(*
    Read and refresh axis parameters
*)
FUNCTION_BLOCK FB_ReadParameterNC IMPLEMENTS I_ReadParameter
VAR
    {attribute 'no_copy'}
    AxisRef : REFERENCE TO AXIS_REF;
	// NC parameters that are exposed with pytmc pragmas
    {attribute 'pytmc' := '
        pv: PLC:AxisPar
        io: i
        field: DESC Axis configuration parameters in the numerical controller.
    '}
    stAxisParametersExposed : ST_AxisParameterSetExposed;
    // MC_ReadParameterSet Output
    fbMcReadParams: MC_ReadParameterSet;
    {attribute 'hide'}
    stAxisParameters: ST_AxisParameterSet;
    {attribute 'hide'}
    NCParamsTimer : TON;
    {attribute 'hide'}
	bExecParamsRead: BOOL;
    {attribute 'hide'}
	bAxisParamsInit: BOOL;
END_VAR

// Periodic update of NC parameters
NCParamsTimer( IN:=NOT bExecParamsRead, PT:=T#1S);

bExecParamsRead S= NCParamsTimer.Q;

fbMcReadParams(
    Parameter:=stAxisParameters,
    Axis:=AxisRef,
    Execute:= bExecParamsRead );

// Copy axis parameters that we want to expose to the EPICS layer.
stAxisParametersExposed.bCtrlEnablePosDiffControl     := stAxisParameters.bCtrlEnablePosDiffControl;
stAxisParametersExposed.bEncEnableSoftEndMaxControl   := stAxisParameters.bEncEnableSoftEndMaxControl;
stAxisParametersExposed.bEncEnableSoftEndMinControl   := stAxisParameters.bEncEnableSoftEndMinControl;
stAxisParametersExposed.fAccelerationMax              := stAxisParameters.fAccelerationMax;
stAxisParametersExposed.fCtrlPosDiffMax               := stAxisParameters.fCtrlPosDiffMax;
stAxisParametersExposed.fCtrlPosDiffMaxTime           := stAxisParameters.fCtrlPosDiffMaxTime;
stAxisParametersExposed.fDecelerationMax              := stAxisParameters.fDecelerationMax;
stAxisParametersExposed.fEncSoftEndMax                := stAxisParameters.fEncSoftEndMax;
stAxisParametersExposed.fEncSoftEndMin                := stAxisParameters.fEncSoftEndMin;
stAxisParametersExposed.fVeloMaximum                  := stAxisParameters.fVeloMaximum;
stAxisParametersExposed.fEncOffset               	  := stAxisParameters.fEncOffset;
stAxisParametersExposed.fEncScaleFactorInternal       := stAxisParameters.fEncScaleFactorInternal;

bExecParamsRead R= fbMcReadParams.Done OR fbMcReadParams.Error;
bAxisParamsInit S= fbMcReadParams.Done;

{warning 'Add property implementation'}
PROPERTY AxisReadParamsInit : BOOL
GET
AxisReadParamsInit := bAxisParamsInit;
END_GET
END_PROPERTY

{warning 'Add property implementation'}
PROPERTY Busy : BOOL
GET
Busy := fbMcReadParams.Busy;
END_GET
END_PROPERTY

METHOD PUBLIC CallAfterInit
VAR_INPUT
    AxisRef : REFERENCE TO AXIS_REF;
END_VAR
THIS^.AxisRef REF= AxisRef;
END_METHOD

{warning 'Add property implementation'}
PROPERTY Done : BOOL
GET
Done := fbMcReadParams.Done;
END_GET
END_PROPERTY

{warning 'Add property implementation'}
PROPERTY Error : BOOL
GET
Error := fbMcReadParams.Error;
END_GET
END_PROPERTY

{warning 'Add property implementation'}
PROPERTY ErrorID : UDINT
GET
ErrorID := fbMcReadParams.ErrorID;
END_GET
END_PROPERTY

//FB_Init is always available implicitly and it is used primarily for initialization.
//The return value is not evaluated. For a specific influence, you can also declare the
//methods explicitly and provide additional code there with the standard initialization
//code. You can evaluate the return value.
METHOD FB_Init: BOOL
VAR_INPUT
    bInitRetains: BOOL; // TRUE: the retain variables are initialized (reset warm / reset cold)
    bInCopyCode: BOOL;  // TRUE: the instance will be copied to the copy code afterward (online change)
    AxisRef : REFERENCE TO AXIS_REF;
END_VAR
THIS^.AxisRef REF= AxisRef;
END_METHOD

{warning 'Add property implementation'}
PROPERTY Message : T_MAXSTRING
GET
END_GET
END_PROPERTY

METHOD ReadParameters
VAR_INPUT
    Enable : BOOL;
    RefreshDelay : TIME;
END_VAR
fbMcReadParams(
    Parameter:=stAxisParameters,
    Axis:=THIS^.AxisRef,
    Execute:= Enable );
	
NCParamsTimer.PT:=RefreshDelay;
END_METHOD

END_FUNCTION_BLOCK

(* stored: Version 1.1.0.1
   POU FB_ReadParameterNC: Id {0a080461-8875-4b57-a673-44abaad03a9d}, SpecialFunc None
   Property AxisReadParamsInit: Id {0109e5c1-4895-4b1a-9b52-46a0b8e2477f}
   Get Get: Id {20a2d9ed-7c9e-44bc-9052-1da3a8039812}
   Property Busy: Id {027c86ab-2c4c-431c-83d3-a5f280a9f4be}
   Get Get: Id {71f3d4a5-5815-498a-9dc2-dd0484d5e903}
   Method CallAfterInit: Id {f18b7d6f-c3da-460b-84aa-32d432fd132a}
   Property Done: Id {e98d6c07-6b86-4458-b10f-56cbec3afbe1}
   Get Get: Id {0b3720d9-74c0-4b42-ab6a-f777060e2826}
   Property Error: Id {48964554-9c0e-4daf-bea2-36931ed4e51d}
   Get Get: Id {c59c9eb4-e912-4bca-ad7b-68b0f66032f4}
   Property ErrorID: Id {530b840d-dfad-4b4f-9afc-f45789cd4abf}
   Get Get: Id {e4b754f9-0ba4-4250-b008-bc6a86a67490}
   Method FB_Init: Id {9a2f321a-6442-4481-94f8-cad0f90b6a8f}
   Property Message: Id {87c74a72-7209-4ca3-a50c-82afcaba9293}
   Get Get: Id {22b2cbd8-48fc-4d7c-b048-86eb05394900}
   Method ReadParameters: Id {7e1988df-13bf-409f-9bba-5c8975b3fe8b} *)
